TYPE ST_AxisInterface :
STRUCT
	INPUT	: ST_AxisIn;
	OUTPUT	: ST_AxisOut;
	
END_STRUCT
END_TYPE

(* stored: Version 1.1.0.1, ProductVersion 3.1.4022.12
   DUT ST_AxisInterface: Id {79e15c89-3aca-498d-862a-00753d1274d2} *)
